// TIA Portal V20 export
// export: Created 2026-07-10T11:12:35.3352414Z, ExportSetting WithDefaults, DisplayName Totally Integrated Automation Portal, DisplayVersion V20, DisplayName TIA Portal Openness, DisplayVersion V20, DisplayName TIA Portal Version Control Interface, DisplayVersion V20, DisplayName STEP 7 Professional, DisplayVersion V20, DisplayName STEP 7 Safety, DisplayVersion V20, DisplayName WinCC Basic/Comfort/Advanced, DisplayVersion V20, DisplayName WinCC Unified, DisplayVersion V20
FUNCTION_BLOCK "ChlorMeasurment"   // FB21, SCL
{ S7_Optimized_Access := 'TRUE' }
VERSION : 0.1
// stored: AutoNumber true, IsIECCheckEnabled false, IsRetainMemResEnabled false, MemoryReserve 100, SetENOAutomatically false, UDAEnableTagReadback false
   VAR_OUTPUT
      blockDosing : Bool;
   END_VAR
   VAR RETAIN
      EnableMeasurment_TON { S7_SetPoint := 'True'} : TON_TIME;
      BlockDosing_TON { S7_SetPoint := 'True'} : TON_TIME;
   END_VAR
   VAR
      enableMeasureTime : Real;
      ChlorationCalculate { S7_SetPoint := 'True'} : "ChlorationCalculate";
      blockDosingTime : Real;
      R_TRIG { S7_SetPoint := 'True'} : R_TRIG;
   END_VAR
   VAR RETAIN
      Initial { S7_SetPoint := 'True'} : Bool := True;
   END_VAR
BEGIN
   IF "MB".Table.CycleDay >= "MB".Table.ChlorMeasureTable[3].CycleDay THEN
       #enableMeasureTime := "MB".Table.ChlorMeasureTable[3].MeasureTime;
       #blockDosingTime := "MB".Table.ChlorMeasureTable[3].BlockTime;
   ELSIF "MB".Table.CycleDay >= "MB".Table.ChlorMeasureTable[2].CycleDay THEN
       #enableMeasureTime := "MB".Table.ChlorMeasureTable[2].MeasureTime;
       #blockDosingTime := "MB".Table.ChlorMeasureTable[2].BlockTime;
   ELSIF "MB".Table.CycleDay >= "MB".Table.ChlorMeasureTable[1].CycleDay THEN
       #enableMeasureTime := "MB".Table.ChlorMeasureTable[1].MeasureTime;
       #blockDosingTime := "MB".Table.ChlorMeasureTable[1].BlockTime;
   ELSIF "MB".Table.CycleDay >= "MB".Table.ChlorMeasureTable[0].CycleDay THEN
       #enableMeasureTime := "MB".Table.ChlorMeasureTable[0].MeasureTime;
       #blockDosingTime := "MB".Table.ChlorMeasureTable[0].BlockTime;
   END_IF;

   #R_TRIG(CLK:="MB".Table.HMI_ChlorModeOn);

   IF #R_TRIG.Q THEN
       #ChlorationCalculate.doseCorection := 1;
       #ChlorationCalculate.doseCorectionOld := 1;
       #Initial := TRUE;
       "MB".Table.MeasureChanged := FALSE;
       RESET_TIMER(#EnableMeasurment_TON);
       RESET_TIMER(#BlockDosing_TON);
   END_IF;


   IF NOT "MB".Table.HMI_ChlorModeOn THEN
       "MB".Table.MeasureChanged := FALSE;
       RESET_TIMER(#EnableMeasurment_TON);
       RESET_TIMER(#BlockDosing_TON);
   END_IF;


   "MB".Table.TimeToMeasure := #enableMeasureTime - DINT_TO_REAL(#EnableMeasurment_TON.ET)/1000/60/60;
   "MB".Table.TimeToBlock := #blockDosingTime - DINT_TO_REAL(#BlockDosing_TON.ET)/1000/60/60;

   #blockDosing := #BlockDosing_TON.Q;
   "MB".Table.MeasureNotEntered := #blockDosing;

   "MB".Table.CriticalMeasureON := FALSE;

   IF "MB".Table.MeasuredChlor >= "MB".Table.CriticalMeasure THEN
       "MB".Table.CriticalMeasureON := TRUE;
       "MB".Table.ChlorationParams.ActualDose := 0;
   END_IF;

   IF "MB".Table.ChangeChlorMeasure THEN
       IF #EnableMeasurment_TON.Q OR #Initial THEN
           "MB".Table.MeasuredChlor := "MB".Table.ChlorMeasuredValue;
           #ChlorationCalculate(ChlorationParams := "MB".Table.ChlorationParams,
                                measuredChlorine := "MB".Table.ChlorMeasuredValue);
           "MB".Table.MeasureChanged := TRUE;
           RESET_TIMER(#EnableMeasurment_TON);
           RESET_TIMER(#BlockDosing_TON);
       END_IF;
       "MB".Table.ChangeChlorMeasure := FALSE;
       #Initial := FALSE;
       #BlockDosing_TON(IN := TRUE,
                        PT := REAL_TO_DINT(#blockDosingTime) * 1000 * 60*60);
       #EnableMeasurment_TON(IN := TRUE,
                             PT := REAL_TO_DINT(#enableMeasureTime) * 1000 * 60*60);
   END_IF;

   IF #EnableMeasurment_TON.Q THEN
       "MB".Table.MeasureChanged := FALSE;
   END_IF;
END_FUNCTION_BLOCK
